(* IEC 61131-3 sources: AXOpen/src/components.kuka.robotics/app/src/IO/PLC_LINE, 2 files *)

(* ---- HwIdentifiers.st ---- *)
TYPE
    HwIdentifiers : WORD
    (
        KRC4_HwID :=	WORD#259,
        KRC4_DIO512_512_digital_in__and_outputs_HwID :=	WORD#262,
        KRC4_KRC4_HwID :=	WORD#261,
        KRC4_KRC4_KRC4_ProfiNet_5_0_HwID :=	WORD#263,
        KRC4_KRC4_profinet_HwID :=	WORD#257,
        KRC4_KRC4_profinet_Port_1_HwID :=	WORD#258,
        KRC4_Rack_HwID :=	WORD#260,
        plc_line_HwID :=	WORD#32,
        plc_line_Rail_0_HwID :=	WORD#264,
        plc_line_plc_line_HwID :=	WORD#48,
        plc_line_plc_line_CPU_display_1_HwID :=	WORD#54,
        plc_line_plc_line_Card_reader_writer_1_HwID :=	WORD#51,
        plc_line_plc_line_DP_interface_1_HwID :=	WORD#60,
        plc_line_plc_line_OPC_UA_1_HwID :=	WORD#117,
        plc_line_plc_line_profinet_x1_HwID :=	WORD#64,
        plc_line_plc_line_profinet_x1_Port_1_HwID :=	WORD#65,
        plc_line_plc_line_profinet_x1_Port_2_HwID :=	WORD#66,
        plc_line_plc_line_profinet_x2_HwID :=	WORD#72,
        plc_line_plc_line_profinet_x2_Port_3_HwID :=	WORD#73,
        plc_line_plc_line_virtual_communication_interface_HwID :=	WORD#135,
        profinet_plc_line_HwID :=	WORD#256,

        NONE := WORD#0
    );
END_TYPE

(* ---- CopyInputs.st ---- *)
FUNCTION CopyInputs
	VAR_EXTERNAL
		HwInputs : HwInputs;
		PlcInputs : PlcInputs;
	END_VAR
	PlcInputs._homeSensor_1	:= HwInputs._homeSensor_1;
	PlcInputs._workSensor_1	:= HwInputs._workSensor_1;
	PlcInputs._homeSensor_2	:= HwInputs._homeSensor_2;
	PlcInputs._workSensor_2	:= HwInputs._workSensor_2;
END_FUNCTION
